PROGRAM PRG_ErrorHandling
VAR
	nErrorBits : UDINT;
	nWarningBits : UDINT;
	
	fbStartUpTimer : TON := (PT := tStartUpTime);
	bStartUpCheck : BOOL;
	bErrorInStartUp : BOOL;
	bErrorInReady : BOOL;
	bErrorInOperational : BOOL;
	bErrorInShutdown : BOOL;
	bAllErrorsAcknowledged : BOOL;
	
	
	
	
	fbEventLogging : FB_EventLogging;
	aSetEventCounterToZero : ARRAY [0..iNumberOfMessages-1] OF USINT;
	n : USINT;
	
	fbSafetyCounter : FB_SafetyCounter;
END_VAR
VAR CONSTANT
	tStartUpTime : TIME := T#10S;
	tSafetyCounterTimeout : TIME := T#5s;
	
	iNumberOfMessages : USINT := 23;			//*set the number of MessageIDs here*
	iNumberOfWarnings : USINT := 16;			//*set the number of Warnings here*
	iNumberOfErrors : USINT := 6;				//*set the number of Errors here*
END_VAR

doSetWarningBits(	nErrorIDServiceModule := PRG_MainController.fbServiceModule.nErrorID,
					nErrorIDLevitationSystem := PRG_MainController.fbLevitationSystem.nErrorID,
					nErrorIDGuidanceSystem := PRG_MainController.fbGuidanceSystem.nErrorID,
					nErrorIDMainController := PRG_ErrorHandling.fbSafetyCounter.nErrorID);
					
doSetErrorBits(		nErrorIDServiceModule := PRG_MainController.fbServiceModule.nErrorID,
					nErrorIDLevitationSystem := PRG_MainController.fbLevitationSystem.nErrorID,
					nErrorIDGuidanceSystem := PRG_MainController.fbGuidanceSystem.nErrorID,
					nErrorIDMainController := PRG_ErrorHandling.fbSafetyCounter.nErrorID);

fbSafetyCounter();
fbEventLogging();

							
CASE PRG_MainController.eState OF
	TopLevelSTM.STARTUP:
		bAllErrorsAcknowledged := FALSE;
		doStartUpCheck(	eConditionServiceModule := PRG_MainController.fbServiceModule.eCondition,
						eConditionLevitationSystem := PRG_MainController.fbLevitationSystem.eCondition,
						eConditionGuidanceSystem := PRG_MainController.fbGuidanceSystem.eCondition);

										
	TopLevelSTM.READY:
		IF nErrorBits <> 0 THEN
			bErrorInReady := TRUE;
		ELSE
			bErrorInReady := FALSE;
		END_IF
		
	TopLevelSTM.OPERATIONAL:
		IF nErrorBits <> 0 THEN
			bErrorInOperational := TRUE;
		ELSE
			bErrorInOperational := FALSE;
		END_IF
		
	TopLevelSTM.SHUTDOWN:
		IF NOT bErrorInOperational THEN
			IF nErrorBits <> 0 THEN
				bErrorInShutdown := TRUE;
			ELSE
				bErrorInShutdown := FALSE;
			END_IF
		END_IF
		
	TopLevelSTM.ERROR:
		IF PRG_MainController.stOperationControlCommands.bAckError THEN
			bErrorInStartUp := FALSE;
			bErrorInReady := FALSE;
			bErrorInOperational := FALSE;
			bErrorInShutdown := FALSE;
			
			//Reset WarningBits and ErrorBits
			nWarningBits := 0;
			nErrorBits := 0;
			
			//Reset Event Logging
			FOR n := 0 TO iNumberOfMessages-1 DO
				aSetEventCounterToZero[n] := 0;
				IF n = iNumberOfMessages-1 THEN
					aSetEventCounterToZero[n] := 1;
				END_IF
			END_FOR
			fbEventLogging.aEventCounter := aSetEventCounterToZero;

			
			bAllErrorsAcknowledged := TRUE;
		END_IF
END_CASE

METHOD PRIVATE doSetErrorBits
VAR_INPUT
	nErrorIDServiceModule : UDINT;
	nErrorIDLevitationSystem : UDINT;
	nErrorIDGuidanceSystem : UDINT;
	nErrorIDMainController : UDINT;
END_VAR
IF PRG_MainController.fbServiceModule.eActivationStatus = ActivationStatus.Disabled THEN
	nErrorIDServiceModule := 0;
END_IF
IF PRG_MainController.fbLevitationSystem.eActivationStatus = ActivationStatus.Disabled THEN
	nErrorIDLevitationSystem := 0;
	nErrorIDMainController.1 := 0;
	nErrorIDMainController.2 := 0;
	nErrorIDMainController.3 := 0;
	nErrorIDMainController.4 := 0;
END_IF
IF PRG_MainController.fbGuidanceSystem.eActivationStatus = ActivationStatus.Disabled THEN
	nErrorIDGuidanceSystem := 0;
	nErrorIDMainController.1 := 0;
	nErrorIDMainController.2 := 0;
	nErrorIDMainController.3 := 0;
	nErrorIDMainController.4 := 0;
END_IF


//ServiceModule

//LevitationSystem

//GuidanceSystem
		
//MainController
nErrorBits.0 := nErrorIDMainController.0;
nErrorBits.1 := nErrorIDMainController.1;
nErrorBits.2 := nErrorIDMainController.2;
nErrorBits.3 := nErrorIDMainController.3;
nErrorBits.4 := nErrorIDMainController.4;
nErrorBits.5 := nErrorIDMainController.5;
END_METHOD

METHOD PRIVATE doSetWarningBits
VAR_INPUT
	nErrorIDServiceModule : UDINT;
	nErrorIDLevitationSystem : UDINT;
	nErrorIDGuidanceSystem : UDINT;
	nErrorIDMainController : UDINT;
END_VAR
IF PRG_MainController.fbServiceModule.eActivationStatus = ActivationStatus.Disabled THEN
	nErrorIDServiceModule := 0;
END_IF
IF PRG_MainController.fbLevitationSystem.eActivationStatus = ActivationStatus.Disabled THEN
	nErrorIDLevitationSystem := 0;
END_IF
IF PRG_MainController.fbGuidanceSystem.eActivationStatus = ActivationStatus.Disabled THEN
	nErrorIDGuidanceSystem := 0;
END_IF

//ServiceModule
nWarningBits.0 := nErrorIDServiceModule.0;
nWarningBits.1 := nErrorIDServiceModule.1;
nWarningBits.2 := nErrorIDServiceModule.2;
nWarningBits.3 := nErrorIDServiceModule.3;
nWarningBits.4 := nErrorIDServiceModule.4;
nWarningBits.5 := nErrorIDServiceModule.5;
nWarningBits.6 := nErrorIDServiceModule.6;
nWarningBits.7 := nErrorIDServiceModule.7;
nWarningBits.8 := nErrorIDServiceModule.8;
nWarningBits.9 := nErrorIDServiceModule.9;

//LevitationSystem
nWarningBits.10 := nErrorIDLevitationSystem.0;
nWarningBits.11 := nErrorIDLevitationSystem.1;

//GuidanceSystem
nWarningBits.12 := nErrorIDGuidanceSystem.0;
nWarningBits.13 := nErrorIDGuidanceSystem.1;
nWarningBits.14 := nErrorIDGuidanceSystem.2;
nWarningBits.15 := nErrorIDGuidanceSystem.3;

//MainController
END_METHOD

METHOD PRIVATE doStartUpCheck
VAR_INPUT
	eConditionServiceModule : HighLevelCondition;
	eConditionLevitationSystem : HighLevelCondition;
	eConditionGuidanceSystem : HighLevelCondition;
END_VAR
IF PRG_MainController.stOperationControlCommands.nOperationMode <> 7 THEN
	IF (eConditionServiceModule = HighLevelCondition.RUN OR eConditionServiceModule = HighLevelCondition.SLEEP) AND (eConditionLevitationSystem = HighLevelCondition.RUN OR eConditionLevitationSystem = HighLevelCondition.SLEEP) AND (eConditionGuidanceSystem = HighLevelCondition.RUN OR eConditionGuidanceSystem = HighLevelCondition.SLEEP) AND NOT (eConditionServiceModule = HighLevelCondition.SLEEP AND eConditionLevitationSystem = HighLevelCondition.SLEEP AND eConditionGuidanceSystem = HighLevelCondition.SLEEP) THEN
		fbStartUpTimer(IN := FALSE);
		bStartUpCheck := TRUE;
	ELSE
		fbStartUpTimer(IN := TRUE);
		IF fbStartUpTimer.Q THEN
			fbStartUpTimer(IN := FALSE);
			bErrorInStartUp := TRUE;
			bStartUpCheck := FALSE;
		ELSE
			bStartUpCheck := FALSE;
		END_IF
	END_IF
ELSE
		fbStartUpTimer(IN := TRUE);
		IF fbStartUpTimer.Q THEN
			fbStartUpTimer(IN := FALSE);
			bErrorInStartUp := TRUE;
			bStartUpCheck := FALSE;
		ELSE
			bStartUpCheck := FALSE;
		END_IF
END_IF
END_METHOD

END_PROGRAM

(* stored: Version 1.1.0.1, ProductVersion 3.1.4024.12
   POU PRG_ErrorHandling: Id {433be138-7b85-46da-b772-f3bde756a423}, SpecialFunc None
   Method doSetErrorBits: Id {7ab45513-1aec-42bb-b9e7-dee8cdaad788}
   Method doSetWarningBits: Id {d18467fe-3cef-435e-aa39-c9f682b69083}
   Method doStartUpCheck: Id {87175268-e8b8-4ec5-8912-ba89808905e0} *)
